// Block: PPrgArchive14

DATA_BLOCK PPrgArchive14
VERSION : 0.1
   NON_RETAIN
   VAR
      PRG : Array[1301..1400] of PPrg_Data;
   END_VAR

BEGIN
   // No initialization required
END_DATA_BLOCK
